(* IEC 61131-3 sources: RL_MAR/experiments/comparison/llm4plc/results/gpt-4o-mini_20260506_100619/20260506_101722, 4 files *)

(* ---- generated_code_iteration_0.st ---- *)
ructured-text
START_ST
FUNCTION_BLOCK GreenhouseWateringSystem
    VAR
        state : INT;                     (* Current state of the system *)
        prevState : INT;                (* Previous state of the system *)
        SoilMoistureSensor : REAL;      (* Input for soil moisture level (0-100%) *)
        SprinklersOn : BOOL := FALSE;    (* Output for controlling sprinklers - on/off *)
        ResponseDelay : TIME := T#5s;   (* Example response delay for the system *)
        LastMoistureReading : REAL;      (* Last recorded soil moisture reading *)
        DelayTimer : TON;                (* Timer for response delay *)
    END_VAR

    (* State Definitions *)
    CONSTANT STATE_INITIALIZE : INT := 0;
    CONSTANT STATE_WAIT : INT := 1;
    CONSTANT STATE_SPRINKLERS_ON : INT := 2;
    CONSTANT STATE_SPRINKLERS_OFF : INT := 3;

    (* Initialization *)
    IF state = STATE_INITIALIZE THEN
        SprinklersOn := FALSE;
        state := STATE_WAIT;  (* Transition to WAIT state after initialization *)
    END_IF

    (* State Machine Logic *)
    CASE state OF
        STATE_WAIT:
            (* Wait for soil moisture reading *)
            LastMoistureReading := SoilMoistureSensor;  (* Update last moisture reading *)
            IF SoilMoistureSensor < 30.0 THEN
                state := STATE_SPRINKLERS_ON;  (* Activate sprinklers if moisture is low *)
            ELSIF SoilMoistureSensor > 70.0 THEN
                state := STATE_SPRINKLERS_OFF;  (* Deactivate sprinklers if moisture is high *)
            END_IF

        STATE_SPRINKLERS_ON:
            SprinklersOn := TRUE;  (* Turn on sprinklers *)
            IF SoilMoistureSensor >= 30.0 THEN
                state := STATE_WAIT;  (* Check moisture level again *)
            END_IF

        STATE_SPRINKLERS_OFF:
            SprinklersOn := FALSE;  (* Turn off sprinklers *)
            IF SoilMoistureSensor <= 70.0 THEN
                state := STATE_WAIT;  (* Check moisture level again *)
            END_IF

    END_CASE

END_FUNCTION_BLOCK
END_ST

(* ---- generated_code_iteration_1.st ---- *)
START_REASON
The errors in the original Structured Text (ST) code occurred due to the incorrect placement of the CONSTANT declarations. In Structured Text, CONSTANTS should be declared within the VAR section, and they should not be placed outside of it. This caused the compiler to throw an error indicating an unexpected token 'CONSTANT'. To resolve this, I will move the CONSTANT declarations into the VAR section and ensure the overall structure adheres to the requirements.
END_REASON

START_ST
FUNCTION_BLOCK GreenhouseWateringSystem
    VAR
        state : INT;                     (* Current state of the system *)
        prevState : INT;                (* Previous state of the system *)
        SoilMoistureSensor : REAL;      (* Input for soil moisture level (0-100%) *)
        SprinklersOn : BOOL := FALSE;    (* Output for controlling sprinklers - on/off *)
        ResponseDelay : TIME := T#5s;   (* Example response delay for the system *)
        LastMoistureReading : REAL;      (* Last recorded soil moisture reading *)
        DelayTimer : TON;                (* Timer for response delay *)

        (* State Definitions *)
        STATE_INITIALIZE : INT := 0;
        STATE_WAIT : INT := 1;
        STATE_SPRINKLERS_ON : INT := 2;
        STATE_SPRINKLERS_OFF : INT := 3;
    END_VAR

    (* Initialization *)
    IF state = STATE_INITIALIZE THEN
        SprinklersOn := FALSE;
        state := STATE_WAIT;  (* Transition to WAIT state after initialization *)
    END_IF

    (* State Machine Logic *)
    CASE state OF
        STATE_WAIT:
            (* Wait for soil moisture reading *)
            LastMoistureReading := SoilMoistureSensor;  (* Update last moisture reading *)
            IF SoilMoistureSensor < 30.0 THEN
                state := STATE_SPRINKLERS_ON;  (* Activate sprinklers if moisture is low *)
            ELSIF SoilMoistureSensor > 70.0 THEN
                state := STATE_SPRINKLERS_OFF;  (* Deactivate sprinklers if moisture is high *)
            END_IF

        STATE_SPRINKLERS_ON:
            SprinklersOn := TRUE;  (* Turn on sprinklers *)
            IF SoilMoistureSensor >= 30.0 THEN
                state := STATE_WAIT;  (* Check moisture level again *)
            END_IF

        STATE_SPRINKLERS_OFF:
            SprinklersOn := FALSE;  (* Turn off sprinklers *)
            IF SoilMoistureSensor <= 70.0 THEN
                state := STATE_WAIT;  (* Check moisture level again *)
            END_IF

    END_CASE

END_FUNCTION_BLOCK
END_ST

(* ---- generated_code_iteration_2.st ---- *)
START_REASON
The errors in the original Structured Text (ST) code occurred due to the use of non-integer values in the CASE statement. In Structured Text, the CASE statement requires the case labels to be of the same type as the variable being evaluated. In this case, the state variable is of type INT, and the case labels must also be integer constants. The previous implementation used variable assignments for state definitions, which may not be recognized as constants in the context of the CASE statement. To resolve this, I will declare the state definitions as constants within the VAR section and ensure they are used correctly in the CASE statement.
END_REASON

START_ST
FUNCTION_BLOCK GreenhouseWateringSystem
    VAR
        state : INT;                     (* Current state of the system *)
        prevState : INT;                (* Previous state of the system *)
        SoilMoistureSensor : REAL;      (* Input for soil moisture level (0-100%) *)
        SprinklersOn : BOOL := FALSE;    (* Output for controlling sprinklers - on/off *)
        ResponseDelay : TIME := T#5s;   (* Example response delay for the system *)
        LastMoistureReading : REAL;      (* Last recorded soil moisture reading *)
        DelayTimer : TON;                (* Timer for response delay *)

        (* State Definitions *)
        STATE_INITIALIZE : INT := 0;
        STATE_WAIT : INT := 1;
        STATE_SPRINKLERS_ON : INT := 2;
        STATE_SPRINKLERS_OFF : INT := 3;
    END_VAR

    (* Initialization *)
    IF state = STATE_INITIALIZE THEN
        SprinklersOn := FALSE;
        state := STATE_WAIT;  (* Transition to WAIT state after initialization *)
    END_IF

    (* State Machine Logic *)
    CASE state OF
        STATE_WAIT:
            (* Wait for soil moisture reading *)
            LastMoistureReading := SoilMoistureSensor;  (* Update last moisture reading *)
            IF SoilMoistureSensor < 30.0 THEN
                state := STATE_SPRINKLERS_ON;  (* Activate sprinklers if moisture is low *)
            ELSIF SoilMoistureSensor > 70.0 THEN
                state := STATE_SPRINKLERS_OFF;  (* Deactivate sprinklers if moisture is high *)
            END_IF

        STATE_SPRINKLERS_ON:
            SprinklersOn := TRUE;  (* Turn on sprinklers *)
            IF SoilMoistureSensor >= 30.0 THEN
                state := STATE_WAIT;  (* Check moisture level again *)
            END_IF

        STATE_SPRINKLERS_OFF:
            SprinklersOn := FALSE;  (* Turn off sprinklers *)
            IF SoilMoistureSensor <= 70.0 THEN
                state := STATE_WAIT;  (* Check moisture level again *)
            END_IF

    END_CASE

END_FUNCTION_BLOCK
END_ST

(* ---- generated_code_iteration_3.st ---- *)
START_REASON
The errors in the original Structured Text (ST) code occurred due to the use of variable assignments for state definitions within the CASE statement. In Structured Text, the CASE statement requires case labels to be integer constants, not variables. To resolve this, I will define the state constants using the `CONST` keyword to ensure they are recognized as constant values. This will allow the CASE statement to function correctly with the defined states.
END_REASON

START_ST
FUNCTION_BLOCK GreenhouseWateringSystem
    VAR
        state : INT;                     (* Current state of the system *)
        prevState : INT;                (* Previous state of the system *)
        SoilMoistureSensor : REAL;      (* Input for soil moisture level (0-100%) *)
        SprinklersOn : BOOL := FALSE;    (* Output for controlling sprinklers - on/off *)
        ResponseDelay : TIME := T#5s;   (* Example response delay for the system *)
        LastMoistureReading : REAL;      (* Last recorded soil moisture reading *)
        DelayTimer : TON;                (* Timer for response delay *)
    END_VAR

    CONST
        STATE_INITIALIZE : INT := 0;     (* State constant for initialization *)
        STATE_WAIT : INT := 1;            (* State constant for waiting *)
        STATE_SPRINKLERS_ON : INT := 2;   (* State constant for sprinklers on *)
        STATE_SPRINKLERS_OFF : INT := 3;   (* State constant for sprinklers off *)
    END_CONST

    (* Initialization *)
    IF state = STATE_INITIALIZE THEN
        SprinklersOn := FALSE;
        state := STATE_WAIT;  (* Transition to WAIT state after initialization *)
    END_IF

    (* State Machine Logic *)
    CASE state OF
        STATE_WAIT:
            (* Wait for soil moisture reading *)
            LastMoistureReading := SoilMoistureSensor;  (* Update last moisture reading *)
            IF SoilMoistureSensor < 30.0 THEN
                state := STATE_SPRINKLERS_ON;  (* Activate sprinklers if moisture is low *)
            ELSIF SoilMoistureSensor > 70.0 THEN
                state := STATE_SPRINKLERS_OFF;  (* Deactivate sprinklers if moisture is high *)
            END_IF

        STATE_SPRINKLERS_ON:
            SprinklersOn := TRUE;  (* Turn on sprinklers *)
            IF SoilMoistureSensor >= 30.0 THEN
                state := STATE_WAIT;  (* Check moisture level again *)
            END_IF

        STATE_SPRINKLERS_OFF:
            SprinklersOn := FALSE;  (* Turn off sprinklers *)
            IF SoilMoistureSensor <= 70.0 THEN
                state := STATE_WAIT;  (* Check moisture level again *)
            END_IF

    END_CASE

END_FUNCTION_BLOCK
END_ST
